FUNCTION_BLOCK ABSTRACT MppcBase EXTENDS TExecution IMPLEMENTS IDevice
VAR_INPUT
END_VAR
VAR_OUTPUT
END_VAR
VAR
	{attribute 'OPC.UA.DA' := '0'}
	_name : STRING;
	{attribute 'OPC.UA.DA' := '0'}
	_deviceID : STRING;					
	{attribute 'OPC.UA.DA' := '0'}
	_family : DeviceFamily;	
	{attribute 'OPC.UA.DA' := '0'}	
	_logger : Logger;
	{attribute 'OPC.UA.DA' := '0'}
	_message : StringBuilder;
	{attribute 'OPC.UA.DA' := '0'}
	_mppcConfig : DeviceConfiguration;
	

END_VAR

PROPERTY DeviceID : STRING
GET
DeviceID := _deviceID;
END_GET
SET
_deviceID := DeviceID;
END_SET
END_PROPERTY

PROPERTY Family : DeviceFamily
GET
Family := _family;
END_GET
SET
_family := Family;
END_SET
END_PROPERTY

PROPERTY Name : STRING
GET
Name := _name;
END_GET
SET
_name := Name;
END_SET
END_PROPERTY

END_FUNCTION_BLOCK

(* stored: Version 1.1.0.1, ProductVersion 3.1.4024.4
   POU MppcBase: Id {094ddfed-9fd7-46cc-98d7-f47b7595877d}, SpecialFunc None
   Property DeviceID: Id {7bfeb1de-77b4-42b1-8fea-62be4722daba}
   Get Get: Id {c5256592-d386-4824-b594-f6e65342ec69}
   Set Set: Id {819f5b00-75f8-4a61-a186-cd3e8539fb52}
   Property Family: Id {5097bb73-f146-457d-9788-3ff66de4a07a}
   Get Get: Id {048954a1-0650-4636-a419-9a4520c838cb}
   Set Set: Id {04a2940c-9e4b-4eb2-afb2-f75672dfcf15}
   Property Name: Id {7c36d05a-1807-4805-92cb-1b939f04d6ba}
   Get Get: Id {8a7e3923-2f10-489f-aae2-f54692da73b8}
   Set Set: Id {fc8c1ef0-60b9-46f5-b16a-e215a96b7e26} *)
